// LS Electric XG5000 project: selfhold
// PLC LSPLC
// module base 0 slot 0: 입출력 모듈:XBC-DR30S (DC 24V 입력 18점, 릴레이 출력 12점)

PROGRAM 자기유지회로 (task: 스캔 프로그램)

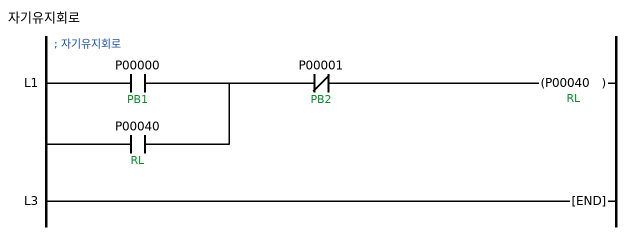
// 자기유지회로
; L1
LOAD      P00000	// PB1
OR        P00040	// RL
AND NOT   P00001	// PB2
OUT       P00040	// RL
; L3
END